PROGRAM TEST_MAIN
VAR
  test_event: TestEvent;
  //test_file_logger: TestFileLogger;
END_VAR

TcUnit.RUN();

END_PROGRAM

(* stored: Version 1.1.0.1, ProductVersion 3.1.4022.18
   POU TEST_MAIN: Id {e0fe771e-7548-4546-bb6c-2059f20a9739}, SpecialFunc None *)
